{attribute 'qualified_only'}
{attribute 'strict'}
TYPE E_CTRL_MODE :
(
	Init := 0,
	Run	:= 10,
	Hold	:= 20,
	Error	:= 9000
);
END_TYPE

(* stored: Version 1.1.0.1, ProductVersion 3.1.4020.12
   DUT E_CTRL_MODE: Id {eb13e7c8-56e2-4a93-8738-0574488b894d} *)
